FUNCTION_BLOCK ReleaseClient
VAR_INPUT
	bReleasePresent : BOOL;
END_VAR

VAR_OUTPUT
	bReleaseAckOut : BOOL;
	bLastHandshakeSuccesful : BOOL;
	bMasterAbortedLastHandshake : BOOL;
END_VAR

VAR
	fbReleasePresentEvent : R_TRIG;
	fbReleaseGoneEvent : F_TRIG;
	fbReleaseAckOutEvent : R_TRIG;
	fbReleaseAckOutGoneEvent : F_TRIG;
END_VAR

fbReleasePresentEvent(CLK:=bReleasePresent);
fbReleaseAckOutEvent(CLK:=bReleaseAckOut);
fbReleaseGoneEvent(CLK:=bReleasePresent);
fbReleaseAckOutGoneEvent(CLK:=bReleaseAckOut);

IF fbReleaseAckOutEvent.Q
THEN
	OnReleaseAckOut();
END_IF

IF fbReleasePresentEvent.Q
THEN
	OnReleasePresent();
END_IF

IF fbReleaseGoneEvent.Q
THEN
	OnReleaseGone();
END_IF

IF fbReleaseAckOutGoneEvent.Q
THEN
	OnHandshakeSuccessful();
END_IF

METHOD OnHandshakeSuccessful : BOOL
VAR_INPUT
END_VAR
bLastHandshakeSuccesful := TRUE;
END_METHOD

METHOD OnReleaseAckOut : BOOL
VAR_INPUT
END_VAR
END_METHOD

METHOD OnReleaseGone : BOOL
VAR_INPUT
END_VAR
IF bReleaseAckOut
THEN
	bReleaseAckOut := FALSE;
ELSE
	bMasterAbortedLastHandshake := TRUE;
END_IF
END_METHOD

METHOD  OnReleasePresent : BOOL
VAR_INPUT
END_VAR
bLastHandshakeSuccesful := FALSE;
bMasterAbortedLastHandshake := FALSE;
END_METHOD

END_FUNCTION_BLOCK

(* stored: Version 1.1.0.1, ProductVersion 3.1.4024.2
   POU ReleaseClient: Id {a80f320d-5687-4adf-b417-42f1f998461e}, SpecialFunc None
   Method OnHandshakeSuccessful: Id {1f77e4dc-7402-4680-8934-e633b7a0b4ce}
   Method OnReleaseAckOut: Id {a8ed3e2b-f776-46b1-82fb-0e25aaf9bcce}
   Method OnReleaseGone: Id {8085a4ea-cd51-4340-8eb0-6a9e5f9472ca}
   Method OnReleasePresent: Id {cbe62dc9-df54-48f1-b145-0ee665cc1735} *)
